// SIMATIC S7-200 SMART project (STEP 7-Micro/WIN SMART), CPU SR40

SYMBOL_TABLE 表格 1
起动按钮             I0.0     // 常开触点
停止按钮             I0.1     // 常开触点
过载               I0.2     // 常开触点
电源               Q0.0     // 电源接触器
短接               Q0.1     // 短接接触器
END_SYMBOL_TABLE

ORGANIZATION_BLOCK MAIN:OB1
TITLE=程序注释：用于初学者的入门例程
BEGIN
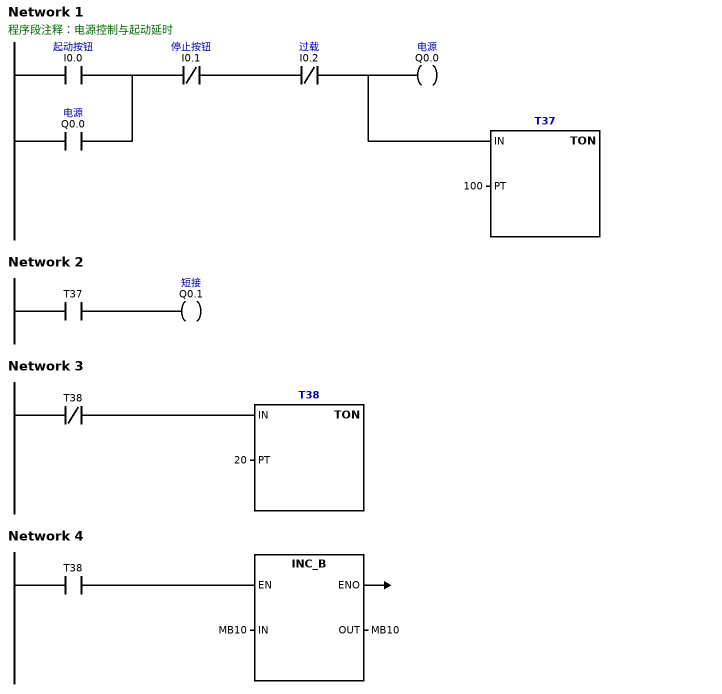
Network 1
// 程序段注释：电源控制与起动延时
LD     起动按钮:I0.0
O      电源:Q0.0
AN     停止按钮:I0.1
AN     过载:I0.2
=      电源:Q0.0
TON    T37, 100
Network 2
LD     T37
=      短接:Q0.1
Network 3
LDN    T38
TON    T38, 20
Network 4
LD     T38
INCB   MB10
END_ORGANIZATION_BLOCK
